FUNCTION_BLOCK E_SWITCH (* Switching (demultiplexing) an event based on boolean input G *)
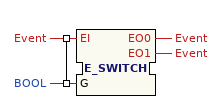
  EVENT_INPUT
    EI WITH G; (* Event Input *)
  END_EVENT
  EVENT_OUTPUT
    EO0; (* Output, switched from EI when G=0 *)
    EO1; (* Output, switched from EI when G=1 *)
  END_EVENT
  VAR_INPUT
    G : BOOL; (* Switch EI to EI0 when G=0, to EI1 when G=1 *)
  END_VAR
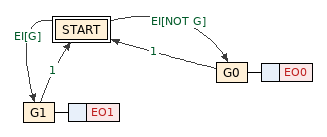
  EC_STATES
    START; (* Initial State *)
    G0 : -> EO0; (* Issue EO0 when EI arrives with G=0 *)
    G1 : -> EO1; (* Issue EO1 when EI arrives with G=1 *)
  END_STATES
  EC_TRANSITIONS
    G0 TO START := 1;
    G1 TO START := 1;
    START TO G0 := EI[NOT G];
    START TO G1 := EI[G];
  END_TRANSITIONS
END_FUNCTION_BLOCK
